{attribute 'qualified_only'}
TYPE JsonElementType :
(
  Undefined := 0,
  Strng,
  Number,
  Object,
  Arry,
  Boolean,
  Null
);
END_TYPE

(* stored: Version 1.1.0.1, ProductVersion 3.1.4024.12
   DUT JsonElementType: Id {3d12cef6-ca69-4d7e-8138-58dc5e3a7e28} *)
